FUNCTION_BLOCK boolMerger (* Basic Function Block Type *)
  (* Standard: 61499-2 *)
  (* Version 0.0, 26/04/2016, Chen-Wei, nxtControl GmbH, Template *)
  PACKAGE Main;
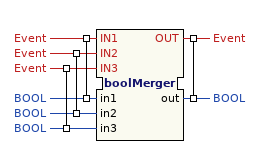
  EVENT_INPUT
    IN1 WITH in1; (* Normal Execution Request *)
    IN2 WITH in2;
    IN3 WITH in3;
  END_EVENT
  EVENT_OUTPUT
    OUT WITH out; (* Execution Confirmation *)
  END_EVENT
  VAR_INPUT
    in1 : BOOL; (* Input event qualifier *)
    in2 : BOOL;
    in3 : BOOL;
  END_VAR
  VAR_OUTPUT
    out : BOOL; (* Output event qualifier *)
  END_VAR
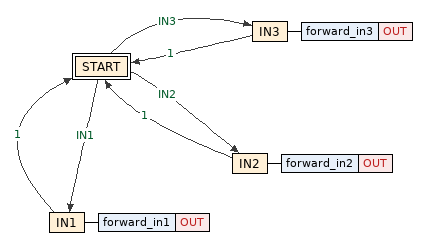
  EC_STATES
    START; (* Initial State *)
    IN1 : forward_in1 -> OUT; (* Normal execution *)
    IN2 : forward_in2 -> OUT;
    IN3 : forward_in3 -> OUT;
  END_STATES
  EC_TRANSITIONS
    START TO IN1 := IN1;
    IN1 TO START := 1;
    START TO IN2 := IN2;
    IN2 TO START := 1;
    START TO IN3 := IN3;
    IN3 TO START := 1;
  END_TRANSITIONS
  ALGORITHM forward_in1 IN ST: (* Normally executed algorithm *)
IN1 := 0;

out := in1;

;
  END_ALGORITHM
  ALGORITHM forward_in2 IN ST:
IN2 := 0;

out := in2;

;
  END_ALGORITHM
  ALGORITHM forward_in3 IN ST:
IN3 := 0;

out := in3;

;
  END_ALGORITHM
END_FUNCTION_BLOCK
